// TIA Portal V20 export
FUNCTION_BLOCK "FB_MainDoorManagement"   // FB510, SCL
{ S7_Optimized_Access := 'TRUE' }
// stored: AutoNumber false, MemoryReserve 100, SetENOAutomatically false
   VAR
      FT_AxisDesactivated { S7_SetPoint := 'True'} : F_TRIG;
      sDoorNotLocked : Bool;
      sLockAutoFrontDoor : Bool;
   END_VAR
BEGIN
   REGION Key[13] Management
       // Key disabled
       "DB_McpKeyboardSignals".sK13_MainDoor.sKeyDisable := NOT "LBP_ModeGroup".E_JOG OR "DB_GestionWorkingModes".sMCP_KxxKeysDisable;

       // Set Door unlock when axis are desactivated
    //   #FTAxisDesactivated(CLK :="DB_DigitalOutputs".Axis_Activation.SWStatus,       WFA A revoir
     //                      Q => "DB_McpKeyboardSignals".K13_MainDoor.KeySWToggleStatus);
   END_REGION

   REGION Unlock / Lock Front Door
       IF "DB_McpKeyboardSignals".sK13_MainDoor.sKeySWTogglePositiveFront
           OR NOT "DB_DataFromSafety".EmergencyStop
           OR "DB_HMISetting".UnlockDoorReq
      //     OR NOT "DB_DigitalOutputs".Axis_Activation.SWStatus       WFA A rajouter 
           OR NOT "DB_DigitalInputs".sFrontDoorClosed.sSWStatus THEN
           "DB_DataToSafety".FrontDoorLock := FALSE;
       ELSIF "DB_McpKeyboardSignals".sK13_MainDoor.sKeySWToggleNegativeFront
           OR #sLockAutoFrontDoor
           OR "DB_HMISetting".LockDoorReq
           AND "DB_DataFromSafety".iFrontDoorClosed
           AND "DB_DigitalInputs".sFrontDoorClosed.sSWStatus THEN
           "DB_DataToSafety".FrontDoorLock := TRUE;
       END_IF;
       "DB_HMISetting".UnlockDoorReq := FALSE;
       "DB_HMISetting".LockDoorReq := FALSE;
   END_REGION

   REGION Led[13] Management
           // OFF : Door Closed and Locked
           // Blink : Door Closed and not Locked
           // ON : Door Open
       "DB_McpKeyboardSignals".sK13_MainDoor.sLedSWStatus :=
       NOT "DB_DataToSafety".FrontDoorLock
       AND ("DB_DataFromSafety".iFrontDoorClosed AND "Clock_1Hz")
       OR NOT "DB_DataFromSafety".iFrontDoorClosed;
   END_REGION

   REGION Alarm messages
       IF NOT "LBP_ModeGroup".E_AUTO THEN
           "LBP_AlarmMsgs".UserA[0].A70UUxx[61] := FALSE;  // Msg: 700061 "Door not locked, cycle start automatically locks main door"
           "LBP_AlarmMsgs".UserA[0].A70UUxx[62] := FALSE;  // Msg: 700062 "Automatic locking of main door on start cycle"
           "LBP_AlarmMsgs".UserA[0].A70UUxx[63] := FALSE;  // Msg: 700063 "Main door open, start cycle not allowed, please close the main door"
       END_IF;

       // Msg: "700061 - Door not locked, cycle start automatically locks main door" 
       "LBP_AlarmMsgs".UserA[0].A70UUxx[61] :=
       NOT "DB_DigitalInputs".sFrontDoorLocked.sSWStatus
       AND "DB_DigitalInputs".sFrontDoorClosed.sSWStatus;

       // Front Door Not Locked
       IF ("DB_DigitalInputs".sFrontDoorLocked.sSWStatus AND #sDoorNotLocked AND "LBP_Chan1".E_ProgRunning)
           OR "MCP1_In".reset THEN
           #sDoorNotLocked := FALSE;
       ELSIF NOT "DB_DigitalInputs".sFrontDoorLocked.sSWStatus AND "DB_DigitalInputs".sFrontDoorClosed.sSWStatus AND "MCP1_In".cycleStart THEN
           #sDoorNotLocked := TRUE;
       END_IF;

       // Msg: 700062 "Automatic locking of main door on start cycle"
       "LBP_AlarmMsgs".UserA[0].A70UUxx[62] := NOT "DB_DigitalInputs".sFrontDoorLocked.sSWStatus AND "DB_DigitalInputs".sFrontDoorClosed.sSWStatus AND ("MCP1_In".cycleStart OR "DB_McpKeyboardSignals".sStartCycle.sKeySWStatus);
       #sLockAutoFrontDoor := "LBP_AlarmMsgs".UserA[0].A70UUxx[62];

       // Msg: 700063 "Main door open, start cycle not allowed, please close the main door"
       IF NOT "DB_DigitalInputs".sFrontDoorLocked.sSWStatus AND NOT "DB_DigitalInputs".sFrontDoorClosed.sSWStatus AND ("MCP1_In".cycleStart OR "DB_McpKeyboardSignals".sStartCycle.sKeySWStatus) THEN
           "LBP_AlarmMsgs".UserA[0].A70UUxx[63] := TRUE;
       ELSIF "DB_DigitalInputs".sFrontDoorClosed.sSWStatus THEN
           "LBP_AlarmMsgs".UserA[0].A70UUxx[63] := FALSE;
       END_IF;
   END_REGION
END_FUNCTION_BLOCK
